# EPICS autosave request: iocs/eigerIOC/iocBoot/iocEiger/auto_settings.req
file "ADBase_settings.req",       P=$(P),  R=cam1:
file "eiger_settings.req",      P=$(P),  R=cam1:
file "NDFile_settings.req",       P=$(P),  R=cam1:
file "NDPluginBase_settings.req", P=$(P),  R=image1:
file "NDStdArrays_settings.req",  P=$(P),  R=image1:
file "commonPlugin_settings.req", P=$(P)
